FUNCTION_BLOCK fb_PTP
VAR_INPUT
END_VAR
VAR_OUTPUT
END_VAR
VAR
	SFCInit : BOOL;
	trn_PosInitDone: BOOL;
	trn_PosPickUpDone: BOOL;
	trn_PosRemoveDone: BOOL;
	trn_PosSampleDone: BOOL;
	trn_PosPocketDone: BOOL;
	fbi_R_TRIG: ARRAY [0..6] OF R_TRIG;
	flg_moveRun: BOOL;
	flg_moveDone: BOOL;
	trn_caluculateDone: BOOL;
	fbi_coordinateCal: fb_coordinateCal;
	fbi_CycleDelayTimer: ARRAY[0..6] OF TON;
	fbi_axisZ_R_TRIG:ARRAY[0..6] OF R_TRIG;
	trn_Mode1Done: BOOL;
	trn_Mode2Done: BOOL;
	var_targetPosX: LREAL;
	var_targetPosY: LREAL;
	var_targetPosZ: LREAL;
	trn_PassPosDone: BOOL;
	trn_SetPosDone: BOOL;
	var_process: INT;
	trn_move_all_done: BOOL;
	var_in_all_pocketNo: INT;
	flg_stop: BOOL;
END_VAR

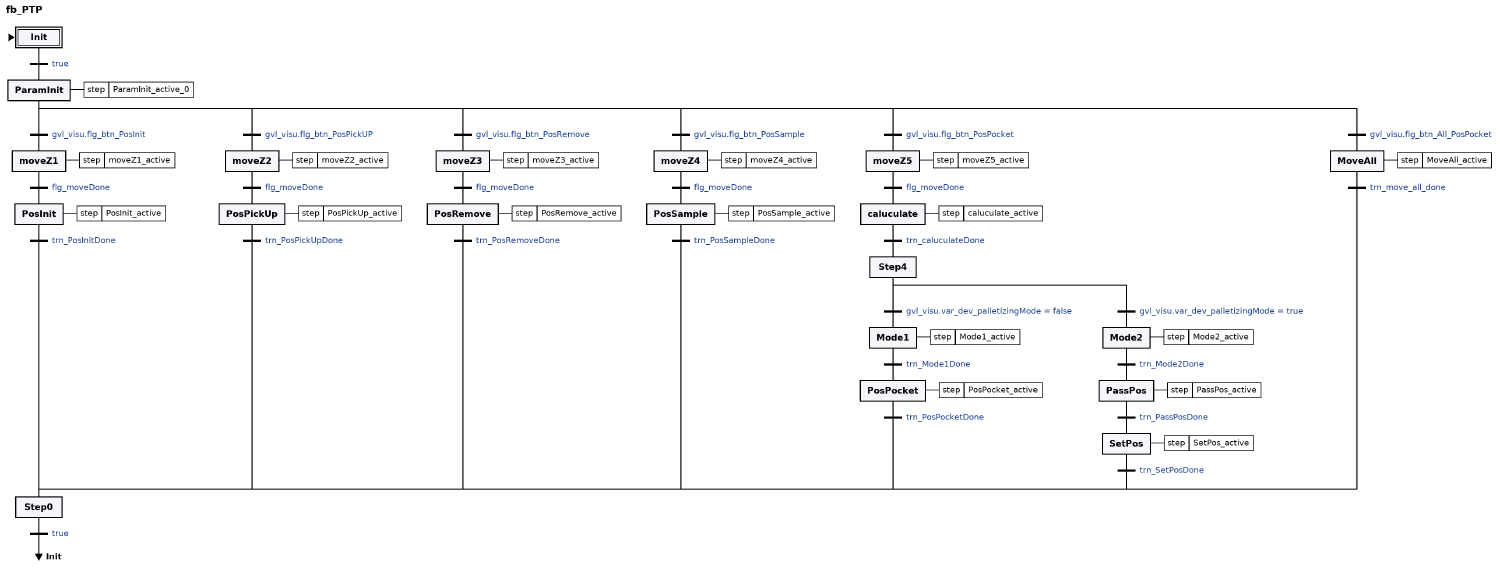
INITIAL_STEP Init:
END_STEP
TRANSITION FROM Init TO ParamInit
    := true;
END_TRANSITION
STEP ParamInit:
    ParamInit_active_0(N);  // step action
END_STEP
TRANSITION FROM ParamInit TO moveZ1
    := gvl_visu.flg_btn_PosInit;
END_TRANSITION
STEP moveZ1:
    moveZ1_active(N);  // step action
END_STEP
TRANSITION FROM moveZ1 TO PosInit
    := flg_moveDone;
END_TRANSITION
STEP PosInit:
    PosInit_active(N);  // step action
END_STEP
TRANSITION FROM PosInit TO Step0
    := trn_PosInitDone;
END_TRANSITION
TRANSITION FROM ParamInit TO moveZ2
    := gvl_visu.flg_btn_PosPickUP;
END_TRANSITION
STEP moveZ2:
    moveZ2_active(N);  // step action
END_STEP
TRANSITION FROM moveZ2 TO PosPickUp
    := flg_moveDone;
END_TRANSITION
STEP PosPickUp:
    PosPickUp_active(N);  // step action
END_STEP
TRANSITION FROM PosPickUp TO Step0
    := trn_PosPickUpDone;
END_TRANSITION
TRANSITION FROM ParamInit TO moveZ3
    := gvl_visu.flg_btn_PosRemove;
END_TRANSITION
STEP moveZ3:
    moveZ3_active(N);  // step action
END_STEP
TRANSITION FROM moveZ3 TO PosRemove
    := flg_moveDone;
END_TRANSITION
STEP PosRemove:
    PosRemove_active(N);  // step action
END_STEP
TRANSITION FROM PosRemove TO Step0
    := trn_PosRemoveDone;
END_TRANSITION
TRANSITION FROM ParamInit TO moveZ4
    := gvl_visu.flg_btn_PosSample;
END_TRANSITION
STEP moveZ4:
    moveZ4_active(N);  // step action
END_STEP
TRANSITION FROM moveZ4 TO PosSample
    := flg_moveDone;
END_TRANSITION
STEP PosSample:
    PosSample_active(N);  // step action
END_STEP
TRANSITION FROM PosSample TO Step0
    := trn_PosSampleDone;
END_TRANSITION
TRANSITION FROM ParamInit TO moveZ5
    := gvl_visu.flg_btn_PosPocket;
END_TRANSITION
STEP moveZ5:
    moveZ5_active(N);  // step action
END_STEP
TRANSITION FROM moveZ5 TO caluculate
    := flg_moveDone;
END_TRANSITION
STEP caluculate:
    caluculate_active(N);  // step action
END_STEP
TRANSITION FROM caluculate TO Step4
    := trn_caluculateDone;
END_TRANSITION
STEP Step4:
END_STEP
TRANSITION FROM Step4 TO Mode1
    := gvl_visu.var_dev_palletizingMode = false;
END_TRANSITION
STEP Mode1:
    Mode1_active(N);  // step action
END_STEP
TRANSITION FROM Mode1 TO PosPocket
    := trn_Mode1Done;
END_TRANSITION
STEP PosPocket:
    PosPocket_active(N);  // step action
END_STEP
TRANSITION FROM PosPocket TO Step0
    := trn_PosPocketDone;
END_TRANSITION
TRANSITION FROM Step4 TO Mode2
    := gvl_visu.var_dev_palletizingMode = true;
END_TRANSITION
STEP Mode2:
    Mode2_active(N);  // step action
END_STEP
TRANSITION FROM Mode2 TO PassPos
    := trn_Mode2Done;
END_TRANSITION
STEP PassPos:
    PassPos_active(N);  // step action
END_STEP
TRANSITION FROM PassPos TO SetPos
    := trn_PassPosDone;
END_TRANSITION
STEP SetPos:
    SetPos_active(N);  // step action
END_STEP
TRANSITION FROM SetPos TO Step0
    := trn_SetPosDone;
END_TRANSITION
TRANSITION FROM ParamInit TO MoveAll
    := gvl_visu.flg_btn_All_PosPocket;
END_TRANSITION
STEP MoveAll:
    MoveAll_active(N);  // step action
END_STEP
TRANSITION FROM MoveAll TO Step0
    := trn_move_all_done;
END_TRANSITION
STEP Step0:
END_STEP
TRANSITION FROM Step0 TO Init
    := true;
END_TRANSITION

ACTION caluculate_active:
IF caluculate._x AND caluculate.x = FALSE THEN
	trn_caluculateDone:= FALSE;
	fbi_coordinateCal.in_flg_run := FALSE;
ELSIF caluculate._x AND caluculate.x THEN
	fbi_coordinateCal.in_flg_run := TRUE;
	IF fbi_coordinateCal.out_flg_Done THEN
		trn_caluculateDone := TRUE;
	END_IF
END_IF

fbi_coordinateCal(
	in_flg_run:= , 
	out_flg_run=> , 
	var_ref_productInfo:= gvl_param.var_productInfo[gvl_param.var_currentProductID], 
	in_var_cavNo:= gvl_visu.var_in_cavNo, 
	in_var_pocketNo:= gvl_visu.var_in_pocketNo, 
	in_var_calculateMode:= , 
	out_flg_busy=> , 
	out_flg_Done=> , 
	out_var_X=> var_targetPosX, 
	out_var_Y=> var_targetPosY, 
	out_var_Z=> var_targetPosZ
);
END_ACTION

ACTION Mode1_active:
IF Mode1._x AND Mode1.x = FALSE THEN
	trn_Mode1Done := FALSE;
	gvl_axis.fbi_motionControler.in_var_targetPosX := var_targetPosX;
	gvl_axis.fbi_motionControler.in_var_targetPosY := var_targetPosY;
	gvl_axis.fbi_motionControler.in_var_targetPosZ := var_targetPosZ;
ELSIF Mode1._x AND Mode1.x THEN
	trn_Mode1Done := TRUE;
END_IF
END_ACTION

ACTION Mode2_active:
IF Mode2._x AND Mode2.x = FALSE THEN
	trn_Mode2Done := FALSE;
	gvl_axis.fbi_motionControler.in_var_targetPosX := var_targetPosX + gvl_param.var_productInfo[gvl_param.var_currentProductID].teachPos.palletize.upperLower[gvl_param.var_currentTrayPos].cav[gvl_visu.var_in_cavNo].teachingDetail.passingPos.x;
	gvl_axis.fbi_motionControler.in_var_targetPosY := var_targetPosY + gvl_param.var_productInfo[gvl_param.var_currentProductID].teachPos.palletize.upperLower[gvl_param.var_currentTrayPos].cav[gvl_visu.var_in_cavNo].teachingDetail.passingPos.y;
	gvl_axis.fbi_motionControler.in_var_targetPosZ := var_targetPosZ + gvl_param.var_productInfo[gvl_param.var_currentProductID].teachPos.palletize.upperLower[gvl_param.var_currentTrayPos].cav[gvl_visu.var_in_cavNo].teachingDetail.passingPos.z;
ELSIF Mode2._x AND Mode2.x THEN
	trn_Mode2Done := TRUE;
END_IF
END_ACTION

ACTION MoveAll_active:
IF MoveAll._x AND MoveAll.x = FALSE THEN
	var_process := 0;
	var_in_all_pocketNo:= 0;
	trn_move_all_done := FALSE;
	gvl_axis.ref_z.Execute := FALSE;
	fbi_coordinateCal.in_flg_run := FALSE;
	gvl_axis.fbi_motionControler.in_flg_start := FALSE;
	flg_stop:= FALSE;
	gvl_visu.flg_All_PosPorket_Move:= FALSE;
ELSIF MoveAll._x AND MoveAll.x THEN
	IF gvl_visu.flg_btn_autoModeStop THEN
		flg_stop:= TRUE;
	END_IF
	CASE var_process OF
		0:
			gvl_axis.ref_z.Position := 50;
			gvl_axis.ref_z.Execute := TRUE;
			fbi_CycleDelayTimer[6].IN := FALSE;
			var_in_all_pocketNo:= var_in_all_pocketNo + 1;
			var_process := 1;
		1:
			gvl_visu.flg_All_PosPorket_Move:= TRUE;
			IF gvl_axis.ref_z.Done THEN
				gvl_axis.ref_z.Execute := FALSE;
				var_process := 2;
			END_IF
		2:
			IF flg_stop THEN
				var_process := 8;
			ELSE
				fbi_coordinateCal.in_flg_run := TRUE;
				gvl_axis.fbi_motionControler.p_Init := TRUE;
				gvl_axis.fbi_motionControler.in_flg_start := FALSE;
				IF fbi_coordinateCal.out_flg_Done THEN
					fbi_coordinateCal.in_flg_run := FALSE;
					var_process := 3;
				END_IF
			END_IF
		3:
			gvl_visu.var_in_pocketNo := var_in_all_pocketNo;
			gvl_axis.fbi_motionControler.p_Init := FALSE;
			gvl_axis.fbi_motionControler.in_var_targetPosX := var_targetPosX;
			gvl_axis.fbi_motionControler.in_var_targetPosY := var_targetPosY;
			gvl_axis.fbi_motionControler.in_var_targetPosZ := var_targetPosZ;
			gvl_axis.fbi_motionControler.in_var_direction := eP_motionDirection.XYZ;
			gvl_axis.fbi_motionControler.in_flg_start := TRUE;
			var_process := 4;
		4:
			IF gvl_axis.fbi_motionControler.out_flg_Done THEN
				gvl_axis.fbi_motionControler.in_flg_start := FALSE;
				var_process := 5;
			END_IF
		5:
			fbi_CycleDelayTimer[6].IN := TRUE;
			var_process := 6;
		6:
			IF fbi_CycleDelayTimer[6].Q THEN
				fbi_CycleDelayTimer[6].IN := FALSE;
				var_process := 7;
			END_IF
		7:
			IF(var_in_all_pocketNo >= gvl_param.var_productInfo[gvl_param.var_currentProductID].pocketSumQty) THEN
				var_process := 8;
			ELSE
				var_process := 0;
			END_IF
		8:	
			gvl_visu.flg_All_PosPorket_Move:= FALSE;
			trn_move_all_done := TRUE;
			
	END_CASE
END_IF
fbi_CycleDelayTimer[6](IN:= , PT:=T#3000MS , Q=> , ET=> );
fbi_coordinateCal(
	in_flg_run:= , 
	out_flg_run=> , 
	var_ref_productInfo:= gvl_param.var_productInfo[gvl_param.var_currentProductID], 
	in_var_cavNo:= gvl_visu.var_in_cavNo, 
	in_var_pocketNo:= var_in_all_pocketNo, 
	in_var_calculateMode:= , 
	out_flg_busy=> , 
	out_flg_Done=> , 
	out_var_X=> var_targetPosX, 
	out_var_Y=> var_targetPosY, 
	out_var_Z=> var_targetPosZ
);
END_ACTION

ACTION moveZ1_active:
IF moveZ1._x AND moveZ1.x = FALSE THEN
	flg_moveDone := FALSE;
	gvl_axis.ref_z.Execute := FALSE;
	gvl_axis.ref_z.Position := 5;
	fbi_axisZ_R_TRIG[0].CLK := FALSE;
ELSIF moveZ1._x AND moveZ1.x THEN
	fbi_axisZ_R_TRIG[0].CLK := TRUE;
	IF gvl_axis.ref_z.Done THEN
		flg_moveDone := TRUE;
	END_IF
END_IF
fbi_axisZ_R_TRIG[0](CLK:= , Q=>gvl_axis.ref_z.Execute );
END_ACTION

ACTION moveZ2_active:
IF moveZ2._x AND moveZ2.x = FALSE THEN
	flg_moveDone := FALSE;
	gvl_axis.ref_z.Execute := FALSE;
	gvl_axis.ref_z.Position := 5;
	fbi_axisZ_R_TRIG[1].CLK := FALSE;
ELSIF moveZ2._x AND moveZ2.x THEN
	fbi_axisZ_R_TRIG[1].CLK := TRUE;
	IF gvl_axis.ref_z.Done THEN
		flg_moveDone := TRUE;
	END_IF
END_IF
fbi_axisZ_R_TRIG[1](CLK:= , Q=>gvl_axis.ref_z.Execute );
END_ACTION

ACTION moveZ3_active:
IF moveZ3._x AND moveZ3.x = FALSE THEN
	flg_moveDone := FALSE;
	gvl_axis.ref_z.Execute := FALSE;
	gvl_axis.ref_z.Position := 5;
	fbi_axisZ_R_TRIG[2].CLK := FALSE;
ELSIF moveZ3._x AND moveZ3.x THEN
	fbi_axisZ_R_TRIG[2].CLK := TRUE;
	IF gvl_axis.ref_z.Done THEN
		flg_moveDone := TRUE;
	END_IF
END_IF
fbi_axisZ_R_TRIG[2](CLK:= , Q=>gvl_axis.ref_z.Execute );
END_ACTION

ACTION moveZ4_active:
IF moveZ4._x AND moveZ4.x = FALSE THEN
	flg_moveDone := FALSE;
	gvl_axis.ref_z.Execute := FALSE;
	gvl_axis.ref_z.Position := 5;
	fbi_axisZ_R_TRIG[3].CLK := FALSE;
ELSIF moveZ4._x AND moveZ4.x THEN
	fbi_axisZ_R_TRIG[3].CLK := TRUE;
	IF gvl_axis.ref_z.Done THEN
		flg_moveDone := TRUE;
	END_IF
END_IF
fbi_axisZ_R_TRIG[3](CLK:= , Q=>gvl_axis.ref_z.Execute );
END_ACTION

ACTION moveZ5_active:
IF moveZ5._x AND moveZ5.x = FALSE THEN
	flg_moveDone := FALSE;
	gvl_axis.ref_z.Execute := FALSE;
	gvl_axis.ref_z.Position := 5;
	fbi_axisZ_R_TRIG[4].CLK := FALSE;
ELSIF moveZ5._x AND moveZ5.x THEN
	fbi_axisZ_R_TRIG[4].CLK := TRUE;
	IF gvl_axis.ref_z.Done THEN
		flg_moveDone := TRUE;
	END_IF
END_IF
fbi_axisZ_R_TRIG[4](CLK:= , Q=>gvl_axis.ref_z.Execute );
END_ACTION

PROPERTY p_init : bool
GET
p_init := THIS^.SFCInit;
END_GET
SET
THIS^.SFCInit := p_init;
END_SET
END_PROPERTY

ACTION ParamInit_active_0:

IF ParamInit._x AND ParamInit.x = FALSE THEN
	gvl_visu.flg_btn_PosInit := FALSE;
	gvl_visu.flg_btn_PosPickUP := FALSE;
	gvl_visu.flg_btn_PosRemove := FALSE;
	gvl_visu.flg_btn_PosSample := FALSE;
	gvl_visu.flg_btn_PosPocket := FALSE;
ELSIF ParamInit._x AND ParamInit.x THEN
	flg_moveDone := FALSE;
END_IF
END_ACTION

ACTION PassPos_active:
IF PassPos._x AND PassPos.x = FALSE THEN
	trn_PassPosDone := FALSE;
	flg_moveRun := FALSE;
	fbi_CycleDelayTimer[5].IN := FALSE;
	gvl_axis.fbi_motionControler.p_Init := TRUE;
	gvl_axis.fbi_motionControler.in_flg_start := FALSE;
	gvl_axis.fbi_motionControler.in_var_direction := eP_motionDirection.XYZ;
ELSIF PassPos._x AND PassPos.x THEN
	gvl_axis.fbi_motionControler.p_Init := FALSE;
	fbi_CycleDelayTimer[5].IN := TRUE;
	IF fbi_CycleDelayTimer[5].Q THEN
		flg_moveRun := TRUE;	
	END_IF
	IF fbi_r_TRIG[5].Q THEN
		gvl_axis.fbi_motionControler.in_flg_start := TRUE;
	END_IF
	IF gvl_axis.fbi_motionControler.out_flg_Done THEN
		trn_PassPosDone := TRUE;
	END_IF
END_IF

fbi_r_TRIG[5](CLK:=flg_moveRun , Q=> );
fbi_CycleDelayTimer[5](IN:= , PT:=T#50MS , Q=> , ET=> );
END_ACTION

ACTION PosInit_active:

IF PosInit._x AND PosInit.x = FALSE THEN
	//flg reset
	trn_PosInitDone := FALSE;
	flg_moveRun := FALSE;
	fbi_CycleDelayTimer[0].IN := FALSE;
	gvl_axis.fbi_motionControler.p_Init := TRUE;
	gvl_axis.fbi_motionControler.in_flg_start := FALSE;
	//insert target postion
	gvl_axis.fbi_motionControler.in_var_targetPosX := gvl_param.var_productInfo[gvl_param.var_currentProductID].teachPos.initial.x;
	gvl_axis.fbi_motionControler.in_var_targetPosY := gvl_param.var_productInfo[gvl_param.var_currentProductID].teachPos.initial.y;
	gvl_axis.fbi_motionControler.in_var_targetPosZ := gvl_param.var_productInfo[gvl_param.var_currentProductID].teachPos.initial.z;
	gvl_axis.fbi_motionControler.in_var_direction := eP_motionDirection.XYZ;
ELSIF PosInit._x AND PosInit.x THEN
	gvl_axis.fbi_motionControler.p_Init := FALSE;
	fbi_CycleDelayTimer[0].IN := TRUE;
	IF fbi_CycleDelayTimer[0].Q THEN
		flg_moveRun := TRUE;
	END_IF
	IF fbi_r_TRIG[0].Q THEN	
		gvl_axis.fbi_motionControler.in_flg_start := TRUE;
	END_IF
	IF gvl_axis.fbi_motionControler.out_flg_Done THEN
		flg_moveRun := FALSE;
		trn_PosInitDone := TRUE;
	END_IF
	
END_IF
fbi_r_TRIG[0](CLK:=flg_moveRun , Q=> );
fbi_CycleDelayTimer[0](IN:= , PT:= T#50MS, Q=> , ET=> );
END_ACTION

ACTION PosPickUp_active:
IF PosPickUp._x AND PosPickUp.x = FALSE THEN
	//flg reset
	trn_PosPickUpDone := FALSE;
	flg_moveRun := FALSE;
	fbi_CycleDelayTimer[1].IN := FALSE;
	gvl_axis.fbi_motionControler.p_Init := TRUE;
	gvl_axis.fbi_motionControler.in_flg_start := FALSE;
	//insert target postion
	gvl_axis.fbi_motionControler.in_var_targetPosX := gvl_param.var_productInfo[gvl_param.var_currentProductID].teachPos.pickUp.x;
	gvl_axis.fbi_motionControler.in_var_targetPosY := gvl_param.var_productInfo[gvl_param.var_currentProductID].teachPos.pickUp.y;
	gvl_axis.fbi_motionControler.in_var_targetPosZ := gvl_param.var_productInfo[gvl_param.var_currentProductID].teachPos.pickUp.z;
	gvl_axis.fbi_motionControler.in_var_direction := eP_motionDirection.XYZ;
ELSIF PosPickUp._x AND PosPickUp.x THEN
	gvl_axis.fbi_motionControler.p_Init := FALSE;
	fbi_CycleDelayTimer[1].IN := TRUE;
	IF fbi_CycleDelayTimer[1].Q THEN
		flg_moveRun := TRUE;
	END_IF
	IF fbi_r_TRIG[1].Q THEN
		gvl_axis.fbi_motionControler.in_flg_start := TRUE;
	END_IF
	IF gvl_axis.fbi_motionControler.out_flg_Done THEN
		trn_PosPickUpDone := TRUE;
	END_IF
END_IF

fbi_r_TRIG[1](CLK:=flg_moveRun , Q=> );
fbi_CycleDelayTimer[1](IN:= , PT:=T#50MS , Q=> , ET=> );
END_ACTION

ACTION PosPocket_active:
IF PosPocket._x AND PosPocket.x = FALSE THEN
	//reset flag
	trn_PosPocketDone := FALSE;
	flg_moveRun := FALSE;
	fbi_CycleDelayTimer[4].IN := FALSE;
	gvl_axis.fbi_motionControler.p_Init := TRUE;
	gvl_axis.fbi_motionControler.in_flg_start := FALSE;
	gvl_axis.fbi_motionControler.in_var_direction := eP_motionDirection.XYZ;
ELSIF PosPocket._x AND PosPocket.x THEN
	gvl_axis.fbi_motionControler.p_Init := FALSE;
	fbi_CycleDelayTimer[4].IN := TRUE;
	IF fbi_CycleDelayTimer[4].Q THEN
		flg_moveRun := TRUE;	
	END_IF
	IF fbi_r_TRIG[4].Q THEN
		gvl_axis.fbi_motionControler.in_flg_start := TRUE;
	END_IF
	IF gvl_axis.fbi_motionControler.out_flg_Done THEN
		trn_PosPocketDone := TRUE;
	END_IF
END_IF

fbi_r_TRIG[4](CLK:=flg_moveRun , Q=> );
fbi_CycleDelayTimer[4](IN:= , PT:=T#50MS , Q=> , ET=> );
END_ACTION

ACTION PosRemove_active:
IF PosRemove._x AND PosRemove.x = FALSE THEN
	//flg reset
	trn_PosRemoveDone := FALSE;
	flg_moveRun := FALSE;
	fbi_CycleDelayTimer[2].IN := FALSE;
	gvl_axis.fbi_motionControler.p_Init := TRUE;
	gvl_axis.fbi_motionControler.in_flg_start := FALSE;
	//insert target postion
	gvl_axis.fbi_motionControler.in_var_targetPosX := gvl_param.var_productInfo[gvl_param.var_currentProductID].teachPos.remove.x;
	gvl_axis.fbi_motionControler.in_var_targetPosY := gvl_param.var_productInfo[gvl_param.var_currentProductID].teachPos.remove.y;
	gvl_axis.fbi_motionControler.in_var_targetPosZ := gvl_param.var_productInfo[gvl_param.var_currentProductID].teachPos.remove.z;
	gvl_axis.fbi_motionControler.in_var_direction := eP_motionDirection.XYZ;
ELSIF PosRemove._x AND PosRemove.x THEN
	gvl_axis.fbi_motionControler.p_Init := FALSE;
	fbi_CycleDelayTimer[2].IN := TRUE;
	IF fbi_CycleDelayTimer[2].Q THEN
		flg_moveRun := TRUE;
	END_IF
	IF fbi_r_TRIG[2].Q THEN
		gvl_axis.fbi_motionControler.in_flg_start := TRUE;
	END_IF
	IF gvl_axis.fbi_motionControler.out_flg_Done THEN
		trn_PosRemoveDone := TRUE;
	END_IF
END_IF

fbi_r_TRIG[2](CLK:=flg_moveRun , Q=> );
fbi_CycleDelayTimer[2](IN:= , PT:=T#50MS , Q=> , ET=> );
END_ACTION

ACTION PosSample_active:
IF PosSample._x AND PosSample.x = FALSE THEN
	//reset flag
	trn_PosSampleDone := FALSE;
	flg_moveRun := FALSE;
	fbi_CycleDelayTimer[3].IN := FALSE;
	gvl_axis.fbi_motionControler.p_Init := TRUE;
	gvl_axis.fbi_motionControler.in_flg_start := FALSE;
	//insert target postion
	gvl_axis.fbi_motionControler.in_var_targetPosX := gvl_param.var_productInfo[gvl_param.var_currentProductID].teachPos.sample[gvl_visu.var_in_sampleCavNo].x;
	gvl_axis.fbi_motionControler.in_var_targetPosX := gvl_param.var_productInfo[gvl_param.var_currentProductID].teachPos.sample[gvl_visu.var_in_sampleCavNo].y;
	gvl_axis.fbi_motionControler.in_var_targetPosX := gvl_param.var_productInfo[gvl_param.var_currentProductID].teachPos.sample[gvl_visu.var_in_sampleCavNo].z;
	gvl_axis.fbi_motionControler.in_var_direction := eP_motionDirection.XYZ;
ELSIF PosSample._x AND PosSample.x THEN
	gvl_axis.fbi_motionControler.p_Init := FALSE;
	fbi_CycleDelayTimer[3].IN := TRUE;
	IF fbi_CycleDelayTimer[3].Q THEN
		flg_moveRun := TRUE;
	END_IF
	IF fbi_r_TRIG[3].Q THEN
		gvl_axis.fbi_motionControler.in_flg_start := TRUE;
	END_IF
	IF gvl_axis.fbi_motionControler.out_flg_Done THEN
		trn_PosSampleDone := TRUE;
	END_IF
END_IF

fbi_r_TRIG[3](CLK:=flg_moveRun , Q=> );
fbi_CycleDelayTimer[3](IN:= , PT:=T#50MS , Q=> , ET=> );
END_ACTION

ACTION SetPos_active:
IF SetPos._x AND SetPos.x = FALSE THEN
	trn_SetPosDone := FALSE;
	var_process := 0;
	gvl_axis.ref_x.Position := var_targetPosX + gvl_param.var_productInfo[gvl_param.var_currentProductID].teachPos.palletize.upperLower[gvl_param.var_currentTrayPos].cav[gvl_visu.var_in_cavNo].teachingDetail.settingPOs.x;
	gvl_axis.ref_y.Position := var_targetPosY + gvl_param.var_productInfo[gvl_param.var_currentProductID].teachPos.palletize.upperLower[gvl_param.var_currentTrayPos].cav[gvl_visu.var_in_cavNo].teachingDetail.settingPOs.y;
	gvl_axis.ref_z.Position := var_targetPosZ + gvl_param.var_productInfo[gvl_param.var_currentProductID].teachPos.palletize.upperLower[gvl_param.var_currentTrayPos].cav[gvl_visu.var_in_cavNo].teachingDetail.settingPOs.z;
ELSIF SetPos._x AND SetPos.x THEN
	CASE var_process OF
		0:
			gvl_axis.ref_x.Execute := TRUE;
			gvl_axis.ref_y.Execute := TRUE;
			gvl_axis.ref_z.Execute := TRUE;
			IF gvl_axis.fbi_mc_absX.Done AND gvl_axis.fbi_mc_absY.Done AND gvl_axis.fbi_mc_absZ.Done THEN
				var_process := 1;
			END_IF
		1:
			gvl_axis.ref_x.Execute := FALSE;
			gvl_axis.ref_y.Execute := FALSE;
			gvl_axis.ref_z.Execute := FALSE;
			trn_SetPosDone := TRUE;
	END_CASE
END_IF
END_ACTION

END_FUNCTION_BLOCK

(* stored: Version 1.1.0.1, ProductVersion 3.1.4024.11
   POU fb_PTP: Id {2e652826-6f0f-4dc7-b660-d15e20414ba1}, SpecialFunc None
   Action caluculate_active: Id {c7aa8955-5437-4f55-bd34-46e74a716597}
   Action Mode1_active: Id {9d7dd620-2a84-4ac9-828b-d5d194bea40f}
   Action Mode2_active: Id {575d719d-dc5d-4827-a44e-0113aa4b49b6}
   Action MoveAll_active: Id {4c2a2b2c-6df4-49e5-96d3-21f867c48dc4}
   Action moveZ1_active: Id {4e9692ca-0658-44cb-b0e1-a3785c4ce4cc}
   Action moveZ2_active: Id {c432afe7-bbc7-417f-903a-34edb87c6dfa}
   Action moveZ3_active: Id {34ec93a3-dcf4-493b-a88e-4cc24637dd62}
   Action moveZ4_active: Id {a5d988df-508b-407b-9cf9-31c52f8c4b75}
   Action moveZ5_active: Id {4d66a992-c469-4940-a460-27721299fb96}
   Property p_init: Id {52ea87a3-da99-45e6-b222-c8047236eb23}
   Get Get: Id {2fc8e0a7-91a5-47e3-a18f-3a3de895fbf4}
   Set Set: Id {dcd0f827-71c6-4df5-8a0a-5ea143d659b0}
   Action ParamInit_active_0: Id {818df57e-f833-48c3-99b3-a7498353dbf4}
   Action PassPos_active: Id {d46e2da0-9697-4007-abd0-bbeb1d489aea}
   Action PosInit_active: Id {31c1d0e0-3689-40c7-bad4-2493963c5f74}
   Action PosPickUp_active: Id {8faa79e7-60c2-4b61-bbb7-73b9cb3c153f}
   Action PosPocket_active: Id {33a80e9d-4ab8-46f4-a3f1-369006f3c708}
   Action PosRemove_active: Id {e6acf63d-ea55-4099-a2b7-cc0b89614ca9}
   Action PosSample_active: Id {d6629494-9ab2-41fe-a3c6-2fcb6d1084a5}
   Action SetPos_active: Id {b5fee515-1222-43fc-9f82-fe96055bc10d} *)
